TYPE CmpConvBreakStopGroupConfig :
STRUCT
	NumberStops: DINT;
	BreakStopDefault: BreakStopConfig;
	BreakStops: ARRAY[1..cBreakStopGroupMaxInstance] OF BreakStopConfig;
END_STRUCT
END_TYPE

(* stored: Version 1.1.0.1, ProductVersion 3.1.4024.6
   DUT CmpConvBreakStopGroupConfig: Id {0aa50655-465d-4f3c-b496-231f01081e53} *)
